// Mitsubishi GX Works2 project: 홀수켜기   PLC: Q02/Q02H

PROGRAM MAIN
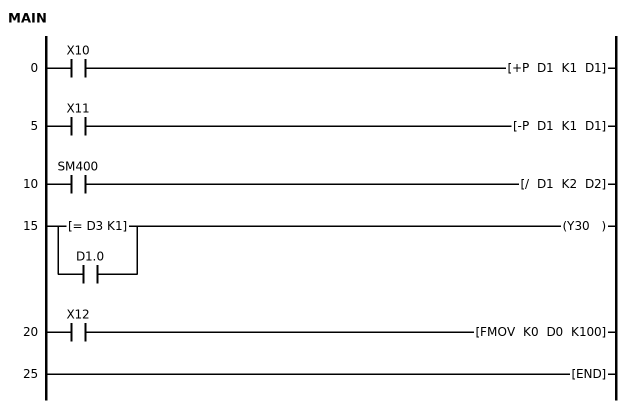
0     LD      X10
      +P      D1 K1 D1
5     LD      X11
      -P      D1 K1 D1
10    LD      SM400
      /       D1 K2 D2
15    LD=     D3 K1
      OR      D1.0
      OUT     Y30
20    LD      X12
      FMOV    K0 D0 K100
25    END
END_PROGRAM
